// TwinCAT 3 PLC project InterfacePractice
// ProgramVersion: 3.1.4024.0
// libraries:
//   Tc2_Standard, * (Beckhoff Automation GmbH)
//   Tc2_System, * (Beckhoff Automation GmbH)
//   Tc3_Module, * (Beckhoff Automation GmbH)
// project tree:
//   / PlcTask.TcTTO
//   POUs/ AddNums.TcPOU, FB_FixedMotor.TcPOU, FB_VariableMotor.TcPOU, FB_VariableSpeedMotor.TcPOU, I_Motor.TcIO, MAIN.TcPOU, MotorController.TcPOU
// (motion and I/O tree: see PLC project functionblockpractice)
// real-time tasks:
//   TASK PlcTask: cycle T#10ms, priority 20, ADS port 350
//   TASK PlcTask2: cycle T#10ms, priority 22, ADS port 352
//   TASK PlcTask1: cycle T#10ms, priority 21, ADS port 351
//   TASK PlcTask3: cycle T#10ms, priority 23, ADS port 353
//   TASK PlcTask4: cycle T#10ms, priority 24, ADS port 354

CONFIGURATION InterfacePractice
    RESOURCE PLC ON TwinCAT3
        TASK PlcTask(INTERVAL := T#10ms, PRIORITY := 22);
        PROGRAM MAIN WITH PlcTask : MAIN;
    END_RESOURCE
END_CONFIGURATION

// ---- POUs/I_Motor.TcIO
INTERFACE I_Motor EXTENDS  __System.IQueryInterface

METHOD Start : BOOL
VAR_INPUT
	
END_VAR
END_METHOD

METHOD Stop : BOOL
VAR_INPUT
	
END_VAR
END_METHOD

END_INTERFACE

// ---- POUs/MAIN.TcPOU
PROGRAM MAIN
VAR
	
	fMotorRunningStatus : BOOL;
	fbFixedMotor1 : FB_FixedMotor;
	iMotor : I_Motor;
	fbVariableMotor1 : FB_VariableMotor;
	
	fbVariableMotor2 : FB_VariableSpeedMotor;
	bRun : BOOL := TRUE;
	
	
	fSpeed : REAL := 34.343;
	bType : BOOL;
	
	fPosition : REAL;;
END_VAR


MotorController(fbFixedMotor1, bRun,fSpeed );
MotorController (fbVariableMotor1, bRun, fSpeed);
MotorController (fbVariableMotor2 , bRun , fSpeed);
fbVariableMotor2.M_SetSpeed(fspeed);
bType := __QUERYINTERFACE(fbVariableMotor2 , iMotor);

END_PROGRAM

// ---- POUs/FB_FixedMotor.TcPOU
FUNCTION_BLOCK FB_FixedMotor IMPLEMENTS I_Motor

VAR
	bRunning : BOOL;
END_VAR

{warning 'add method implementation '}
METHOD Start : BOOL
bRunning := TRUE;
Start := bRunning;
END_METHOD

{warning 'add method implementation '}
METHOD Stop : BOOL
bRunning := FALSE;
Stop := NOT bRunning;
END_METHOD

END_FUNCTION_BLOCK

// ---- POUs/FB_VariableMotor.TcPOU
FUNCTION_BLOCK FB_VariableMotor IMPLEMENTS I_Motor

VAR
	bRunning : BOOL;
END_VAR

{warning 'add method implementation '}
METHOD Start : BOOL
Start := bRunning := TRUE;
END_METHOD

{warning 'add method implementation '}
METHOD Stop : BOOL
bRunning := FALSE;
Stop := NOT bRunning;
END_METHOD

END_FUNCTION_BLOCK

// ---- POUs/FB_VariableSpeedMotor.TcPOU
FUNCTION_BLOCK FB_VariableSpeedMotor EXTENDS FB_VariableMotor

VAR
	fMotorSpeed : REAL;
	fMotorPosition : REAL;
	Trans_CylinderExtended: INT;
	i_bSensorEnd: INT;
	i_bSensorHome: INT;
END_VAR

PROPERTY PUBLIC fPosition : REAL
GET
fPosition := fMotorPosition;
END_GET
SET // PRIVATE
fMotorPosition := fPosition;
END_SET
END_PROPERTY

METHOD M_SetSpeed : BOOL
VAR_INPUT
	fSpeedPercent : REAL;
END_VAR
fMotorSpeed := fSpeedPercent;
M_SetSpeed := TRUE;
END_METHOD

END_FUNCTION_BLOCK

// ---- POUs/MotorController.TcPOU
FUNCTION MotorController : BOOl
VAR_INPUT
	iMotor1 : I_Motor;
	bRun : BOOL;
	fSpeed : REAL;
END_VAR
VAR
END_VAR


IF bRun THEN
	iMotor1.Start();
ELSE
	iMotor1.Stop();
END_IF

END_FUNCTION

// ---- POUs/AddNums.TcPOU
FUNCTION AddNums : INT
VAR_INPUT
	pNum : POINTER TO INT;
END_VAR
VAR
	ppNum : POINTER TO POINTER TO INT;
END_VAR


ppNum := ADR(pNum);
ppNum^^ := 25;

END_FUNCTION
